PROGRAM POU_Mando
VAR
END_VAR

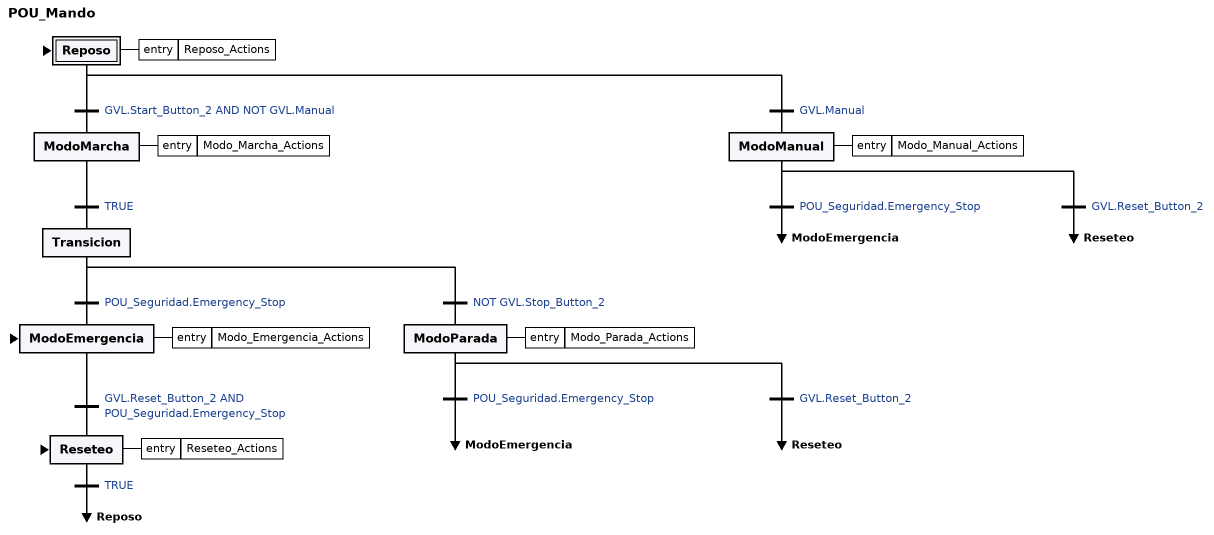
INITIAL_STEP Reposo:
    Reposo_Actions(P1);  // entry action
END_STEP
TRANSITION FROM Reposo TO ModoMarcha
    := GVL.Start_Button_2 AND NOT GVL.Manual;
END_TRANSITION
STEP ModoMarcha:
    Modo_Marcha_Actions(P1);  // entry action
END_STEP
TRANSITION FROM ModoMarcha TO Transicion
    := TRUE;
END_TRANSITION
TRANSITION FROM Reposo TO ModoManual
    := GVL.Manual;
END_TRANSITION
STEP ModoManual:
    Modo_Manual_Actions(P1);  // entry action
END_STEP
TRANSITION FROM ModoManual TO ModoEmergencia
    := POU_Seguridad.Emergency_Stop;
END_TRANSITION
TRANSITION FROM ModoManual TO Reseteo
    := GVL.Reset_Button_2;
END_TRANSITION
STEP Transicion:
END_STEP
TRANSITION FROM Transicion TO ModoEmergencia
    := POU_Seguridad.Emergency_Stop;
END_TRANSITION
STEP ModoEmergencia:
    Modo_Emergencia_Actions(P1);  // entry action
END_STEP
TRANSITION FROM ModoEmergencia TO Reseteo
    := GVL.Reset_Button_2 AND POU_Seguridad.Emergency_Stop;
END_TRANSITION
TRANSITION FROM Transicion TO ModoParada
    := NOT GVL.Stop_Button_2;
END_TRANSITION
STEP ModoParada:
    Modo_Parada_Actions(P1);  // entry action
END_STEP
TRANSITION FROM ModoParada TO ModoEmergencia
    := POU_Seguridad.Emergency_Stop;
END_TRANSITION
TRANSITION FROM ModoParada TO Reseteo
    := GVL.Reset_Button_2;
END_TRANSITION
STEP Reseteo:
    Reseteo_Actions(P1);  // entry action
END_STEP
TRANSITION FROM Reseteo TO Reposo
    := TRUE;
END_TRANSITION

ACTION Desactivar_Alarmas_Actions:
//Se desactivan las alarmas
GVL.Alarm_Siren  := FALSE;
GVL.Warning_Light  := FALSE;
GVL.Factory_IO_Pause := FALSE;
END_ACTION

ACTION Modo_Emergencia_Actions:
GVL.Marcha := FALSE; // Se indica que la planta no puede funcionar
END_ACTION

ACTION Modo_Manual_Actions:
// Se indica mediante una luz que el siguiente botón a pulsar sería el de Reset
GVL.Start_Button_2_Light := FALSE;
GVL.Reset_Button_2_Light := TRUE;
END_ACTION

ACTION Modo_Marcha_Actions:
GVL.Marcha := TRUE; // Se indica que la planta puede comenzar a funcionar
GVL.Emitter_1 := TRUE; // Se activa la emisión de piezas
GVL.Belt_Conveyor_2m_1 := 1; // Se activa la cinta de entrada
// Se indica mediante una luz que el siguiente botón a pulsar sería el de Stop
GVL.Start_Button_2_Light := FALSE; 
GVL.Stop_Button_2_Light := TRUE;
END_ACTION

ACTION Modo_Parada_Actions:
GVL.Emitter_1 := FALSE; // Se desactiva la emisión de piezas
GVL.Belt_Conveyor_2m_1 := 0; // Se desactiva la cinta de entrada
// Se indica mediante una luz que el siguiente botón a pulsar sería el de Reset
GVL.Stop_Button_2_Light := FALSE; 
GVL.Reset_Button_2_Light := TRUE;
END_ACTION

ACTION Reposo_Actions:
GVL.Marcha := FALSE; // Se indica que la planta no puede funcionar
// Se indica mediante una luz que el siguiente botón a pulsar sería el de Start
GVL.Start_Button_2_Light := TRUE; 
GVL.Reset_Button_2_Light := FALSE;
// Se permite que la planta se mueva dentro del factory I/O
GVL.Factory_IO_Pause := FALSE;
GVL.Factory_IO_Reset := FALSE;
END_ACTION

ACTION Reseteo_Actions:
GVL.Factory_IO_Reset := TRUE;
POU_Reset_Planta();
GVL.Manual := FALSE;
//Se desactivan las alarmas
//GVL.Alarm_Siren  := FALSE;
//GVL.Warning_Light  := FALSE;
END_ACTION

END_PROGRAM

(* stored: Version 1.1.0.1, ProductVersion 3.1.4024.12
   POU POU_Mando: Id {680136ca-075c-4e14-baab-2aee1a722adf}, SpecialFunc None
   Action Desactivar_Alarmas_Actions: Id {ddfa02ba-e0b2-4364-b878-731b6c75f73d}
   Action Modo_Emergencia_Actions: Id {afd2d41b-57c3-41c9-abcd-a1b3d1c32e42}
   Action Modo_Manual_Actions: Id {e1a04f41-03fd-4b6b-a057-558686dfa31d}
   Action Modo_Marcha_Actions: Id {4ff40a7b-c953-49fd-9ebb-8f6e6257cfdf}
   Action Modo_Parada_Actions: Id {8b9e64b5-1ae5-4e79-b6ab-878700fcfe92}
   Action Reposo_Actions: Id {3b9c9df1-1504-46a3-96bf-248a11775764}
   Action Reseteo_Actions: Id {93f7e9bb-60db-4dfe-934d-f3b5a963c776} *)
